FUNCTION SclBytePNP : BYTE
VAR_INPUT
	byUnscaled	: BYTE;
END_VAR
VAR
END_VAR

IF byUnscaled = 0 THEN
	SclBytePNP	:= 0;
ELSE
	SclBytePNP	:= 255;
END_IF

END_FUNCTION

(* stored: Version 1.1.0.1, ProductVersion 3.1.4024.6
   POU SclBytePNP: Id {9e36fe55-d402-4065-ab28-8572f72e7b29}, SpecialFunc None *)
